// TIA Portal V17 export
// export: Created 2023-12-22T15:28:36.8494994Z, ExportSetting WithDefaults, DisplayName Totally Integrated Automation Portal, DisplayVersion V17, DisplayName TIA Portal Openness, DisplayVersion V17, DisplayName TIA Portal Version Control Interface, DisplayVersion V17, DisplayName STEP 7 Professional, DisplayVersion V17, DisplayName STEP 7 Safety, DisplayVersion V17, DisplayName WinCC Advanced, DisplayVersion V17
DATA_BLOCK "DIx_1_DB"   // DB200
VERSION : 0.1
// stored: AutoNumber false, DBAccessibleFromOPCUA true, InstanceOfName DIx_1, InstanceOfType FB
"DIx_1"
   // VAR RETAIN
   //    AllBlock { S7_SetPoint := 'True'} : "DI_ex";
   //    signal_2 { S7_SetPoint := 'True'} : "DI_ex";
   //    signal_3 { S7_SetPoint := 'True'} : "DI_ex";
   //    signal_4 { S7_SetPoint := 'True'} : "DI_ex";
   //    signal_5 { S7_SetPoint := 'True'} : "DI_ex";
   //    signal_6 { S7_SetPoint := 'True'} : "DI_ex";
   //    signal_7 { S7_SetPoint := 'True'} : "DI_ex";
   //    signal_8 { S7_SetPoint := 'True'} : "DI_ex";
   //    signal_9 { S7_SetPoint := 'True'} : "DI_ex";
   //    signal_10 { S7_SetPoint := 'True'} : "DI_ex";
   //    signal_11 { S7_SetPoint := 'True'} : "DI_ex";
   //    signal_12 { S7_SetPoint := 'True'} : "DI_ex";
   //    Time_DTL { S7_SetPoint := 'True'} : DTL;
   // END_VAR
BEGIN
END_DATA_BLOCK
